% RSLogix 500 project I2P JOB 21 - ALEXANDER_LOYND_BAK104.RSS, saved by version 10.00.00.00 %
PROJECT "ML06A"    % processor: Bul.1763 MicroLogix 1100 Series B %

PROGRAM FILES
  LAD 2   5 rungs

DATA FILES
  O0 OUTPUT  4 elements
  I1 INPUT  6 elements
  S2 STATUS  66 elements
  B3 BINARY  1 elements
  T4 TIMER  1 elements
  C5 COUNTER  1 elements
  R6 CONTROL  1 elements
  N7 INTEGER  1 elements
  F8 FLOAT  1 elements

LADDER 2
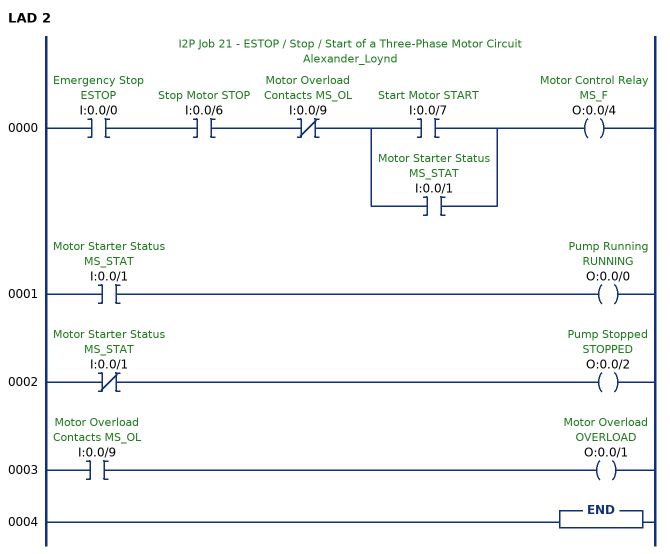
% Rung: 0 %
% I2P Job 21 - ESTOP / Stop / Start of a Three-Phase Motor Circuit
% Alexander_Loynd %
SOR XIC I:0.0/0 XIC I:0.0/6 XIO I:0.0/9 BST XIC I:0.0/7 NXB XIC I:0.0/1 BND OTE O:0.0/4 EOR
%   I:0.0/0  ESTOP  "Emergency Stop" %
%   I:0.0/6  STOP  "Stop Motor" %
%   I:0.0/9  MS_OL  "Motor Overload Contacts" %
%   I:0.0/7  START  "Start Motor" %
%   I:0.0/1  MS_STAT  "Motor Starter Status" %
%   O:0.0/4  MS_F  "Motor Control Relay" %
% Rung: 1 %
SOR XIC I:0.0/1 OTE O:0.0/0 EOR
%   I:0.0/1  MS_STAT  "Motor Starter Status" %
%   O:0.0/0  RUNNING  "Pump Running" %
% Rung: 2 %
SOR XIO I:0.0/1 OTE O:0.0/2 EOR
%   I:0.0/1  MS_STAT  "Motor Starter Status" %
%   O:0.0/2  STOPPED  "Pump Stopped" %
% Rung: 3 %
SOR XIC I:0.0/9 OTE O:0.0/1 EOR
%   I:0.0/9  MS_OL  "Motor Overload Contacts" %
%   O:0.0/1  OVERLOAD  "Motor Overload" %
% Rung: 4 %
SOR END EOR

OTHER DOCUMENTED ADDRESSES
  B3:0/0  ESTOP_STOP_BIT  "Estop/stop info bit"
  B3:0/1  FWD_BIT  "Forward direction bit"
  B3:0/2  REV_BIT  "Reverse direction bit"
  B3:0/3  LAST_FWD  "Motor Last In Forward"
  B3:0/4  LAST_REV  "Motor Last In Reverse"
  I:0.0/2  DIR_STAT  "Control Relay Two Contacts"
  I:0.0/3  MODE_ON  "On Setting 3PSS"
  I:0.0/4  MODE_AUTO  "AUTO Setting 3PSS"
  I:0.0/5  OFF_AUTO  "Off or Auto"
  I:0.0/8  REV  "Start Motor in reverse"
  MOV  
  O:0.0/3  FULL  "Tank Full"
  O:0.0/5  CR2  "Direction Control Relay"
  PB1  "Start Motor"
  T4:0  TIME_ON_DELAY  "Keeps motor stopped when switching to forward/reverse"
  T4:0/DN  T4
  T4:0/TT  MOTOR_CHANGE_TIMER  "Timer for motor change"

DATA TABLE (non-zero values as saved)
DATA T4
% .PRE .ACC %
% T4:0 % 16 0
DATA C5
% .PRE .ACC %
% C5:0 % 16 3
